FUNCTION _LEN : UDINT
VAR_INPUT
	pSrc 	 : POINTER TO BYTE;
	u32Max : UDINT;
END_VAR

	
	_len := 0;

	WHILE (pSrc^ <> 0 and _len < u32Max) DO
		_len := _len+1;
		pSrc := pSrc+1;
	END_WHILE

END_FUNCTION

(* stored: Version 1.1.0.1, ProductVersion 3.1.4024.13
   POU _LEN: Id {49524f06-7335-4cbd-a109-2925dfa8cbc4}, SpecialFunc None *)
